FUNCTION_BLOCK ABSTRACT LightBase EXTENDS TExecution IMPLEMENTS IDevice
VAR_INPUT
END_VAR
VAR_OUTPUT
END_VAR
VAR
	{attribute 'OPC.UA.DA' := '0'}
	_name : STRING;
	{attribute 'OPC.UA.DA' := '0'}
	_deviceID : STRING;				
	{attribute 'OPC.UA.DA' := '0'}	
	_family : DeviceFamily;	
	{attribute 'OPC.UA.DA' := '0'}
	_logger : Logger;
	{attribute 'OPC.UA.DA' := '0'}
	_message : StringBuilder;
	{attribute 'OPC.UA.DA' := '0'}
	_lightConfig : DeviceConfiguration;	
	
	{attribute 'OPC.UA.DA' := '0'}
	_lifeTimeCount : UINT;
	{attribute 'OPC.UA.DA' := '0'}
	_notifyIsAlive : BOOL;
	{attribute 'OPC.UA.DA' := '0'}
	_pulseIsAliveGenerator : TON;				
		
	StateMsg : STRING(255);
	IsAliveMsg : STRING(255);
END_VAR

// Check if it's still alive	
IF _notifyIsAlive THEN
	IsAliveMsg := TO_STRING(_lifeTimeCount);
	_notifyIsAlive := FALSE;
END_IF

IF HardwareGlobalVariables.LightState <> State THEN
	HardwareGlobalVariables.LightState := State;
	StateMsg := ANY_TO_STRING(State);		
END_IF

MessageSchedulerBase();

PROPERTY DeviceID : STRING
GET
DeviceID := _deviceID;
END_GET
SET
_deviceID := DeviceID;
END_SET
END_PROPERTY

PROPERTY Family : DeviceFamily
GET
Family := _family;
END_GET
SET
_family := Family;
END_SET
END_PROPERTY

METHOD IsAlive
VAR_INPUT
END_VAR
_notifyIsAlive := TRUE;

IF _lifeTimeCount < 5 THEN
	_lifeTimeCount := _lifeTimeCount + 1;
ELSE
	_lifeTimeCount := 1;
END_IF
END_METHOD

METHOD MessageSchedulerBase
VAR_INPUT
END_VAR
IF _pulseIsAliveGenerator.Q THEN
	_pulseIsAliveGenerator(IN := FALSE, PT := T#10MS);
		
	IsAlive();	
ELSE
	_pulseIsAliveGenerator(IN := TRUE, PT := T#1000MS);		
END_IF
END_METHOD

PROPERTY Name : STRING
GET
Name := _name;
END_GET
SET
_name := Name;
END_SET
END_PROPERTY

METHOD ABSTRACT SetIntensity
VAR_INPUT
	Execute : BOOL;
	LightId : STRING;
	Intensity : LREAL;
END_VAR
END_METHOD

END_FUNCTION_BLOCK

(* stored: Version 1.1.0.1, ProductVersion 3.1.4024.12
   POU LightBase: Id {65614fd1-6fc9-46bf-8601-806094071640}, SpecialFunc None
   Folder Commands: Id {dd5af989-5b9a-4a4b-a020-56886f985841}
   Property DeviceID: Id {6bd756f4-cedc-4988-82dd-c223d8d02ee3}
   Get Get: Id {f642b7fb-b2de-428a-b05f-2cb86a6d0562}
   Set Set: Id {6ad482d1-1ac9-4159-9124-e7806b9e54f1}
   Property Family: Id {15287f51-1ec6-4cf5-89f5-b89db4d4fdd4}
   Get Get: Id {3913feb6-e8f5-47d6-8a61-27a49ea81f02}
   Set Set: Id {178194f5-bea2-4f64-9707-610d9bd5bf16}
   Method IsAlive: Id {e02d2bd8-0b7c-47f6-b925-1a7553a685a7}
   Method MessageSchedulerBase: Id {e9563ba8-4fb2-42ea-8662-45c6d04194aa}
   Property Name: Id {e71c8f13-9bc0-42a6-9c5c-4c7a18795d93}
   Get Get: Id {085a6715-4abc-4cee-abf8-3d27ba383840}
   Set Set: Id {8bea579d-5fd9-427f-906f-cbba143c2f51}
   Method SetIntensity: Id {f57a947b-6804-42d7-9f21-66a7ec9bb44c} *)
